// TIA Portal project "shorting by weight" (V15)
// Vorlageprojekt für das Buch mit Zielsystem S7-1200

(* hardware
DEVICE "S7-1200-Station_1"  S7-1200 Station
   slot 0: "Baugruppenträger_0"  Rack  V1.0
   slot 1: "PLC_1"  CPU 1211C DC/DC/DC  6ES7 211-1AE40-0XB0  V4.1
DEVICE "HMI_1"  KTP700 Basic PN
   slot 0: "HMI_1"  KTP700 Basic PN  6AV2 123-2GB03-0AX0  15.0.0.0
   slot 1: "HMI_RT_1"  KTP700 Basic PN  6AV2 123-2GB03-0AX0  15.0.0.0
   slot 5: "HMI_1.IE_CP_1"  PROFINET Interface  15.0.0.0
      slot 1: "PROFINET Interface_1"  PROFINET Interface
         slot 1: "Port_1"  Port
*)

// ===== PLC "PLC_1"  CPU 1211C DC/DC/DC =====

VAR_GLOBAL   // PLC tag table "Standard-Variablentabelle"
   "start" AT %I1.0 : Bool;
   "stop" AT %I1.1 : Bool;
   "firstsensor" AT %I0.0 : Bool;
   "atscale" AT %I0.1 : Bool;
   "entryconveyor" AT %Q0.0 : Bool;
   "scaleconveyor" AT %Q0.1 : Bool;
   "leftconveyor" AT %Q0.2 : Bool;
   "rightconveyor" AT %Q0.3 : Bool;
   "frontconveyor" AT %Q0.4 : Bool;
   "sendforward" AT %Q0.5 : Bool;
   "sendright" AT %Q0.6 : Bool;
   "sendleft" AT %Q0.7 : Bool;
   "Tag_1" AT %M0.0 : Bool;
   "Tag_2" AT %M0.1 : Bool;
   "Tag_3" AT %ID30 : Real;
   "Tag_4" AT %M0.2 : Bool;
   "Tag_5" AT %MB30 : Byte;
   "left exit" AT %I0.2 : Bool;
   "right exit" AT %I0.3 : Bool;
   "front exit" AT %I0.4 : Bool;
   "Tag_6" AT %M0.3 : Bool;
   "left count" AT %QD30 : DInt;
   "forward count" AT %QD34 : DInt;
   "right count" AT %QD38 : DInt;
   "weight on screen" AT %QD42 : DInt;
   "Tag_7" AT %M0.4 : Bool;
   "Tag_8" AT %M0.5 : Bool;
   "Reset" AT %I1.2 : Bool;
   "emerg stop" AT %I1.3 : Bool;
END_VAR

DATA_BLOCK "varoi"   // DB1
{ S7_Optimized_Access := 'TRUE' }
VERSION : 0.1
   VAR
      weight : Array[0..2] of Real;
   END_VAR
BEGIN
END_DATA_BLOCK

// folder: System blocks/Program resources

DATA_BLOCK "IEC_Counter_0_DB"   // DB4
{ S7_Optimized_Access := 'TRUE' }
AUTHOR : Simatic
FAMILY : IEC
NAME : CNTR
VERSION : 1.0
// stored: InstanceOfName IEC_COUNTER
"IEC_COUNTER"
BEGIN
END_DATA_BLOCK

// folder: (top level)

FUNCTION "StartConveyor" : Void   // FC1, LAD
{ S7_Optimized_Access := 'TRUE' }
VERSION : 0.1
   VAR_INPUT
      start : Bool;
      stop : Bool;
      "emergency stop" : Bool;
   END_VAR
   VAR_OUTPUT
      "entry conveyor" : Bool;
      "scale conveyor" : Bool;
      "left conveyor" : Bool;
      "right conveyor" : Bool;
      "front conveyor" : Bool;
      "send forward" : Bool;
   END_VAR
BEGIN

REGION Network 1
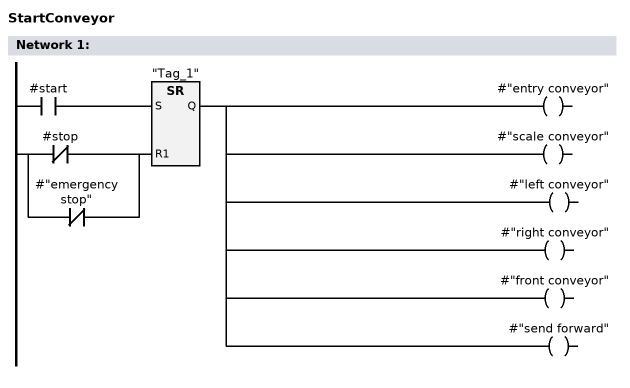
   RUNG wire#powerrail
      Contact( #start )
      S_SR(operand := "Tag_1", r1 := wire#w1)
      wire#w2
      Coil( #"entry conveyor" )
   END_RUNG
   RUNG wire#powerrail
      I_Contact( #stop )
   END_RUNG wire#w1
   RUNG wire#powerrail
      I_Contact( #"emergency stop" )
   END_RUNG wire#w1
   RUNG wire#w2
      Coil( #"scale conveyor" )
   END_RUNG
   RUNG wire#w2
      Coil( #"left conveyor" )
   END_RUNG
   RUNG wire#w2
      Coil( #"right conveyor" )
   END_RUNG
   RUNG wire#w2
      Coil( #"front conveyor" )
   END_RUNG
   RUNG wire#w2
      Coil( #"send forward" )
   END_RUNG
   // the same network as SCL:
   IF #start THEN
       "Tag_1" := TRUE;   // SR flip-flop
   END_IF;
   IF NOT #stop OR NOT #"emergency stop" THEN "Tag_1" := FALSE; END_IF;
   #"entry conveyor" := "Tag_1";
   #"scale conveyor" := "Tag_1";
   #"left conveyor" := "Tag_1";
   #"right conveyor" := "Tag_1";
   #"front conveyor" := "Tag_1";
   #"send forward" := "Tag_1";
END_REGION
END_FUNCTION

FUNCTION "wheeldirection" : Void   // FC2, SCL
{ S7_Optimized_Access := 'TRUE' }
VERSION : 0.1
   VAR_INPUT
      recipe : Int;   // select the recipe (0,1,2)
      "counter" : Int;   // timi pou exei o counter
      weight : Real;   // metroumeno varos
      at_scale : Bool;
   END_VAR
   VAR_OUTPUT
      left : Bool;
      right : Bool;
      weight_display : DInt;
      temp : Array[0..2] of Real;   // temporary table
   END_VAR
   VAR_TEMP
      sort : Array[0..5] of Bool;
   END_VAR
BEGIN
   CASE #recipe OF
       0:
           #sort[0] := 0;
           #sort[1] := 0;
           #sort[2] := 0;
           #sort[3] := 1;
           #sort[4] := 1;
           #sort[5] := 0;
       1:  
           #sort[0] := 0;
           #sort[1] := 1;
           #sort[2] := 1;
           #sort[3] := 0;
           #sort[4] := 0;
           #sort[5] := 0;
       2:
           #sort[0] := 1;
           #sort[1] := 0;
           #sort[2] := 0;
           #sort[3] := 0;
           #sort[4] := 0;
           #sort[5] := 1;
       ELSE
           #recipe := 0;


   END_CASE;


   IF #at_scale = 1 THEN
       #temp[#counter] := #weight;
   END_IF;
   //katefthinsi analoga me to varos. ta varoi sto factory i/o paizoun arketa gia ayto 
   //ekana me toso megalo keno tis times.
   //(parola ayta kinite swsta analoga to metroymeno varos)

   //big boxes
   IF #temp [#counter]> 6.4 AND #temp [#counter] < 8.5 THEN
       #left := #sort[0];
       #right := #sort[1];
   END_IF;
   //medium boxes
   IF #temp [#counter]> 4.5 AND #temp [#counter] < 6.4 THEN
       #left := #sort[2];
       #right := #sort[3];
   END_IF;
   //small boxes
   IF #temp[#counter] > 3.0 AND #temp[#counter] < 4.5 THEN
       #left := #sort[4];
       #right := #sort[5];
   END_IF;
   //------------------------------
   #weight_display := REAL_TO_DINT(#weight);
END_FUNCTION

FUNCTION "counter" : Void   // FC3, LAD
{ S7_Optimized_Access := 'TRUE' }
VERSION : 0.1
   VAR_TEMP   // added for the SCL form of the ladder/FBD networks
      _w1 : Bool;
   END_VAR
BEGIN

REGION Network 1
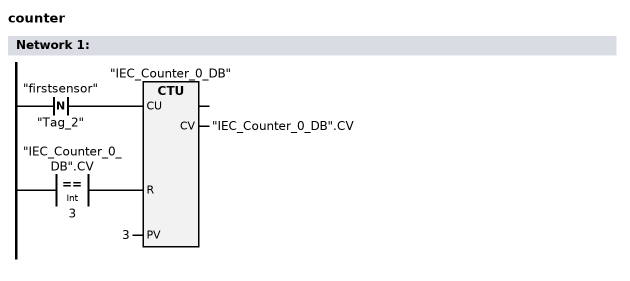
   #_w1 := NOT "firstsensor" AND "Tag_2";   // falling edge of "firstsensor"
   "Tag_2" := "firstsensor";
   "IEC_Counter_0_DB".CTU(CU := #_w1, R := "IEC_Counter_0_DB".CV = 3, PV := 3, CV => "IEC_Counter_0_DB".CV);
END_REGION
END_FUNCTION

FUNCTION "count blocks" : Void   // FC4, LAD
{ S7_Optimized_Access := 'TRUE' }
VERSION : 0.1
   VAR_TEMP   // added for the SCL form of the ladder/FBD networks
      _w1 : Bool;
      _w2 : Bool;
      _w3 : Bool;
   END_VAR
BEGIN

REGION Network 1
   // deixnei stis othones ston pinaka posa koutia perasan
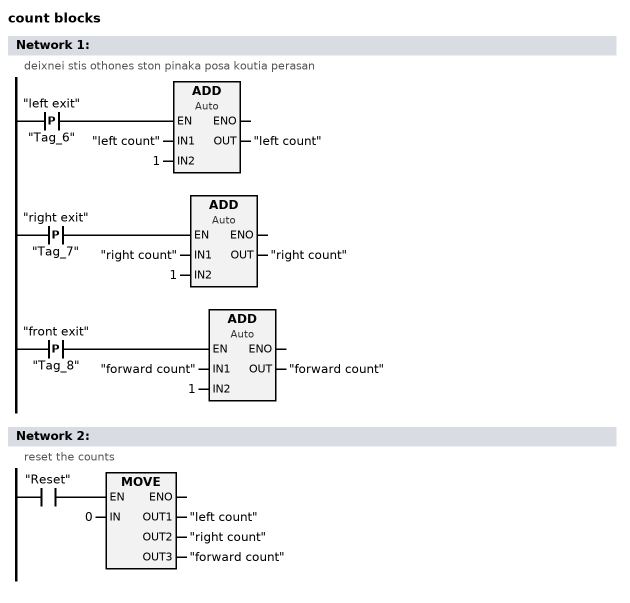
   RUNG wire#powerrail
      P_Contact(operand := "left exit", bit := "Tag_6")
      Add(in1 := "left count", in2 := 1, out => "left count")
   END_RUNG
   RUNG wire#powerrail
      P_Contact(operand := "right exit", bit := "Tag_7")
      Add(in1 := "right count", in2 := 1, out => "right count")
   END_RUNG
   RUNG wire#powerrail
      P_Contact(operand := "front exit", bit := "Tag_8")
      Add(in1 := "forward count", in2 := 1, out => "forward count")
   END_RUNG
   // the same network as SCL:
   #_w1 := "left exit" AND NOT "Tag_6";   // rising edge of "left exit"
   "Tag_6" := "left exit";
   IF #_w1 THEN "left count" := "left count" + 1; END_IF;
   #_w2 := "right exit" AND NOT "Tag_7";   // rising edge of "right exit"
   "Tag_7" := "right exit";
   IF #_w2 THEN "right count" := "right count" + 1; END_IF;
   #_w3 := "front exit" AND NOT "Tag_8";   // rising edge of "front exit"
   "Tag_8" := "front exit";
   IF #_w3 THEN "forward count" := "forward count" + 1; END_IF;
END_REGION

REGION Network 2
   // reset the counts
   RUNG wire#powerrail
      Contact( "Reset" )
      Move(in := 0, out1 => "left count", out2 => "right count", out3 => "forward count")
   END_RUNG
   // the same network as SCL:
   IF "Reset" THEN
       "left count" := 0;
       "right count" := 0;
       "forward count" := 0;
   END_IF;
END_REGION
END_FUNCTION

FUNCTION "MHJ-PLC-Lab-Function-S71200" : Void   // FC9000, SCL
{ S7_Optimized_Access := 'TRUE' }
VERSION : 0.1
   VAR_TEMP
      rdTimeReturn : Int;
      outputTime : DTL;
      SyncVal : Byte;
      forVal : Int;
      forVal_2 : Int;
      Value : Byte;
   END_VAR
   VAR CONSTANT
      CompVal : Byte := 16#34;
      Value_01 : Byte := 16#11;
      Value_01_DW : DWord := 16#A165_D992;
      Value_02_DW : DWord := 16#58BE_4401;
   END_VAR
BEGIN

   #Value:=PEEK(area := 16#82,
        dbNumber := 0,
        byteOffset := 511);
   #Value := #Value + 1;

   POKE(area := 16#82,
        dbNumber := 0,
        byteOffset := 511,
        value := #Value);

   POKE(area:=16#81,
        dbNumber:=0,
        byteOffset:=1016,
        value:=#Value_01_DW);
   POKE(area := 16#81,
        dbNumber := 0,
        byteOffset := 1020,
        value := #Value_02_DW);

   POKE(area := 16#81,
        dbNumber := 0,
        byteOffset := 511,
        value := B#16#00);

   FOR #forVal := 0 TO 120 DO
       FOR #forVal_2:=0 TO 10 DO
           #rdTimeReturn:=RD_SYS_T(#outputTime);
           #rdTimeReturn := WR_SYS_T(#outputTime);
           #rdTimeReturn := RD_SYS_T(#outputTime);
           #rdTimeReturn := WR_SYS_T(#outputTime);
       END_FOR;
       #SyncVal:= PEEK(area := 16#81,
                      dbNumber := 0,
                      byteOffset := 511);
       IF #SyncVal = #CompVal THEN
          GOTO M_1;
       END_IF;
   END_FOR;
   RETURN;

   M_1:
   POKE(area := 16#81,
        dbNumber := 0,
        byteOffset := 511,
        value := B#16#0);
END_FUNCTION

ORGANIZATION_BLOCK "Main"   // OB1, FBD, ProgramCycle
TITLE = "Main Program Sweep (Cycle)"
{ S7_Optimized_Access := 'TRUE' }
VERSION : 0.1
   VAR_INPUT
      Initial_Call : Bool;   // Initial call of this OB
      Remanence : Bool;   // =True, if remanent data are available
   END_VAR
   VAR_TEMP   // added for the SCL form of the ladder/FBD networks
      _w1 : Bool;
   END_VAR
BEGIN

REGION Network 1: Konnektierungsbaustein für PLC-Lab
   // Im Netzwerk 1 wird der Konnektierungsbaustein für PLC-Lab aufgerufen.
   // Dieser Aufruf darf nicht entfernt werden!
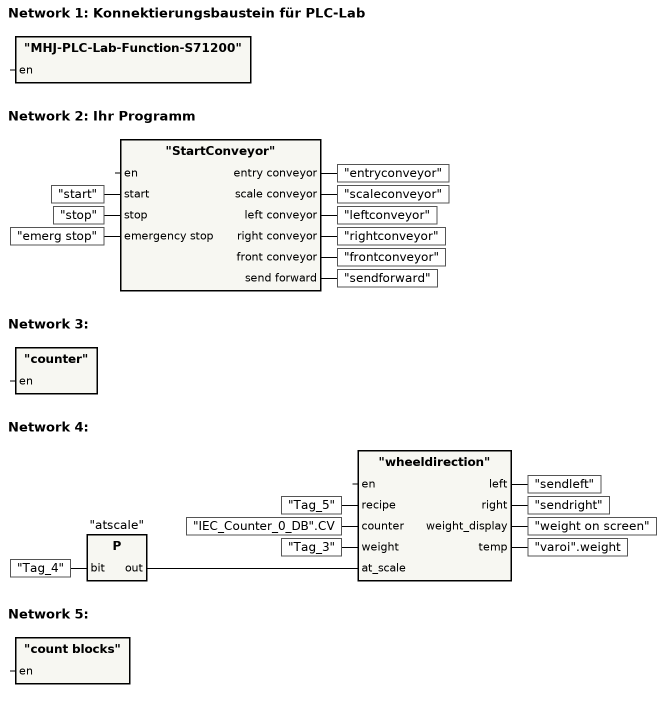
   "MHJ-PLC-Lab-Function-S71200"();
END_REGION

REGION Network 2: Ihr Programm
   // Schreiben Sie ab Netzwerk 2 Ihr Programm
   "StartConveyor"(start := "start",
                   stop := "stop",
                   "emergency stop" := "emerg stop",
                   "entry conveyor" => "entryconveyor",
                   "scale conveyor" => "scaleconveyor",
                   "left conveyor" => "leftconveyor",
                   "right conveyor" => "rightconveyor",
                   "front conveyor" => "frontconveyor",
                   "send forward" => "sendforward");
END_REGION

REGION Network 3
   "counter"();
END_REGION

REGION Network 4
   #_w1 := "atscale" AND NOT "Tag_4";   // rising edge of "atscale"
   "Tag_4" := "atscale";
   "wheeldirection"(recipe := "Tag_5",
                    "counter" := "IEC_Counter_0_DB".CV,
                    weight := "Tag_3",
                    at_scale := #_w1,
                    left => "sendleft",
                    right => "sendright",
                    weight_display => "weight on screen",
                    temp => "varoi".weight);
END_REGION

REGION Network 5
   "count blocks"();
END_REGION
END_ORGANIZATION_BLOCK

(* ===== HMI "HMI_RT_1" =====
system functions are stored by id; their names below are inferred from use
connection "HMI_Connection_1": ETHERNET, SMART_S7_1200_OMS

HMI tags "Default tag table"
   "Tag_ScreenNumber" : UInt, internal
   "Tag_5" : Byte = PLC Tag_5 AT %MB30, 1 s
   "entryconveyor" : Bool = PLC entryconveyor AT %Q0.0, 1 s

text list "Text_list_1": 0 'RECIPE 0'; 1 'RECIPE 1'; 2 'RECIPE 2'

Template "Template_1" 800x480
   Button "Exit" at 714,429 size 71x50; TextOff 'Exit'; PictureOff "ExitRuntime_KTP700_Basic_PN_TR"; PictureOn "ExitRuntime_KTP700_Basic_PN_TR"
      on Release: StopRuntime(0)
   Button "Template_Button" at 614,429 size 71x50; TextOff 'Text'
   Button "Template_Button_1" at 514,429 size 71x50; TextOff 'Text'
   Button "Template_Button_2" at 414,429 size 71x50; TextOff 'Text'
   Button "Template_Button_3" at 314,429 size 71x50; TextOff 'Text'
   Button "Template_Button_4" at 214,429 size 71x50; TextOff 'Text'
   Button "Template_Button_5" at 114,429 size 71x50; TextOff 'Text'
   Button "Start screen" at 14,429 size 71x50; TextOff 'Start screen'; PictureOff "NavigateHome_KTP700_Basic_PN_TR"; PictureOn "NavigateHome_KTP700_Basic_PN_TR"
      on Release: ActivateScreen("Root screen", 0)
   SymbolicIOField "Symbolic_IO_Field_Screen" at 93,9 size 600x33; TextOff '0'; TextOn '1'; TextList "TextList_ScreenNames"
      ProcessValue <- "Tag_ScreenNumber"
      on Change: ActivateScreenByNumber("Tag_ScreenNumber", 0)
   DateTimeField "HmiScreenItemData" at 695,25 size 105x25
   DateTimeField "HmiScreenItemData_1" at 695,0 size 105x25
   GraphicView "Logo" at 0,0 size 91x51; Picture "Logo of HMI_1"

screen "Root screen" 800x480, template "Template_1"
   on GenerateScreen: SetTag("Tag_ScreenNumber", 1)
   SymbolicIOField "Symbolic I/O field_1" at 274,75 size 219x63; TextOff '0'; TextOn '1'; TextList "Text_list_1"
      ProcessValue <- "Tag_5"
      on Activate: function_b3f726e6("Tag_5", 0)
   Rectangle "Rectangle_1" at 85,338 size 69x88
      Appearance <- "Tag_5"
   Rectangle "Rectangle_2" at 338,338 size 69x88
      Appearance <- "Tag_5"
   Rectangle "Rectangle_3" at 617,338 size 69x88
      Appearance <- "Tag_5"
   Rectangle "Rectangle_6" at 0,290 size 85x48
      Appearance <- "Tag_5"
   Rectangle "Rectangle_11" at 617,206 size 69x88
      Appearance <- "Tag_5"
   Rectangle "Rectangle_12" at 338,206 size 69x88
      Appearance <- "Tag_5"
   Rectangle "Rectangle_4" at 85,208 size 69x88
      Appearance <- "Tag_5"
   Rectangle "Rectangle_5" at 152,291 size 85x48
      Appearance <- "Tag_5"
   Rectangle "Rectangle_7" at 253,291 size 85x48
      Appearance <- "Tag_5"
   Rectangle "Rectangle_8" at 407,291 size 85x48
      Appearance <- "Tag_5"
   Rectangle "Rectangle_9" at 533,290 size 85x48
      Appearance <- "Tag_5"
   Rectangle "Rectangle_10" at 686,291 size 85x48
      Appearance <- "Tag_5"
   TextField "Text field_2" at 15,301 size 48x23; Text 'small'
      Appearance <- "Tag_5"
   TextField "Text field_1" at 346,232 size 48x23; Text 'small'
      Appearance <- "Tag_5"
   TextField "Text field_3" at 703,301 size 48x23; Text 'small'
      Appearance <- "Tag_5"
   TextField "Text field_4" at 93,236 size 51x23; Text 'Large'
      Appearance <- "Tag_5"
   TextField "Text field_5" at 421,301 size 51x23; Text 'Large'
      Appearance <- "Tag_5"
   TextField "Text field_6" at 549,296 size 51x23; Text 'Large'
      Appearance <- "Tag_5"
   TextField "Text field_7" at 163,301 size 69x23; Text 'Medium'
      Appearance <- "Tag_5"
   TextField "Text field_8" at 255,301 size 69x23; Text 'Medium'
      Appearance <- "Tag_5"
   TextField "Text field_9" at 618,239 size 69x23; Text 'Medium'
      Appearance <- "Tag_5"
   TextField "Text field_10" at 93,372 size 48x23; Text 'Entry'
      Appearance <- "Tag_5"
   TextField "Text field_11" at 346,371 size 48x23; Text 'Entry'
      Appearance <- "Tag_5"
   TextField "Text field_12" at 627,371 size 48x23; Text 'Entry'
      Appearance <- "Tag_5"
   TextField "Text field_13" at 63,155 size 121x35; Text 'RECIPE 0'
   TextField "Text field_14" at 320,155 size 121x35; Text 'RECIPE 1'
   TextField "Text field_15" at 588,155 size 121x35; Text 'RECIPE 2'
   TextField "Text field_16" at 306,43 size 156x30; Text 'Choose Recipe'
   TextField "Text field_18" at 63,75 size 119x23; Text '= RECIPE OFF'
   TextField "Text field_19" at 63,110 size 113x23; Text '= RECIPE ON'
*)